(* CoDeSys 2.3.9.62 project: EjemploBiestableLD.pro *)
(* Libraries: Standard.lib 4.10.05 10:14:46, IecSfc.lib 2.6.14 10:37:46 *)

(* Global variable list: Global_Variables *)
VAR_GLOBAL
   (* Entradas *)
   Enciende1 : BOOL;
   Apaga1 : BOOL;
  Enciende2 : BOOL;
   Apaga2 : BOOL;
   (*Salidas*)
   Luz1: BOOL;
   Luz2:BOOL;
END_VAR

(* POU PLC_PRG, LD *)
PROGRAM PLC_PRG
VAR

END_VAR
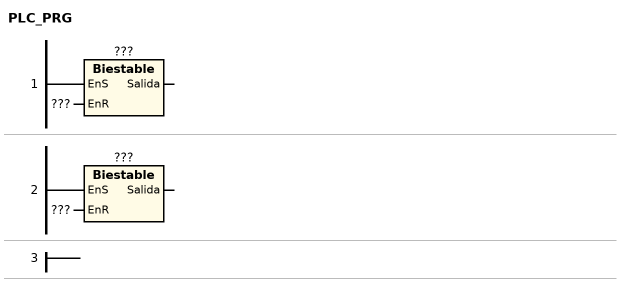
_LD_ (* Ladder Diagram *)
NETWORK 1
	???:Biestable(EnS: *, EnR: ???)
NETWORK 2
	???:Biestable(EnS: *, EnR: ???)
NETWORK 3
	*
_END_LD_
END_PROGRAM

(* POU Biestable, LD *)
FUNCTION_BLOCK Biestable
VAR_INPUT
	EnS: BOOL;
	EnR: BOOL;
END_VAR
VAR_OUTPUT
	Salida: BOOL;
END_VAR
VAR
END_VAR
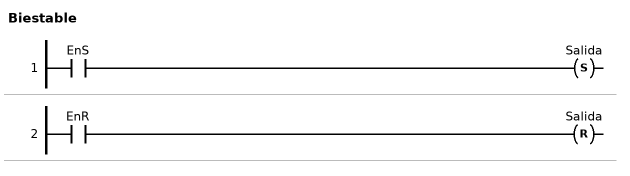
_LD_ (* Ladder Diagram *)
NETWORK 1
	[EnS] --- (S Salida)
NETWORK 2
	[EnR] --- (R Salida)
_END_LD_
(* the same logic as Structured Text *)
(* Network 1 *)
IF EnS THEN Salida := TRUE; END_IF;
(* Network 2 *)
IF EnR THEN Salida := FALSE; END_IF;
END_FUNCTION_BLOCK

(* Visualisation Biestable
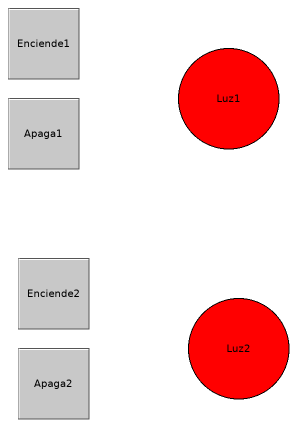
button at (90,30)-(161,101): text "Enciende1"; taps Enciende1
button at (90,120)-(161,191): text "Apaga1"; taps Apaga1
ellipse at (260,70)-(361,171): text "Luz1"; alarm colour if Luz1
button at (100,280)-(171,351): text "Enciende2"; taps Enciende2
button at (100,370)-(171,441): text "Apaga2"; taps Apaga2
ellipse at (270,320)-(371,421): text "Luz2"; alarm colour if Luz2
*)
